(* Logix 5000 project; controller IF2_DEMO Emulate 5570 rev 20.12; software revision 20.04; part 6 of 8 *)
(* tags used below, declared in another part *)
   Alarm_RapidMixStopped : ALARM_DIGITAL;
   CIPSteps : DINT;
   Complete_Manual_Step_AUTO : TIMER;
   Main : MotionVars;
   Mixer_Step_6_AUTORESET : TIMER;
   repeatCIP : BOOL;
   Restart_CIP_Timer_AUTO : TIMER;
   ChangeOver_In_Progress : BOOL;
   Current_Order : STRING;
   DispenserLine : LineData;
   Filler_Stopped : BOOL;
   InitializeDelay : TIMER;
   Labeler_Stopped : BOOL;
   LastOrderCount : DINT;
   LastOrderNumber : STRING;
   ManualCompleted : BOOL;
   MixAgitatorDelayTimer : TIMER;
   MIXCIPStep_DelayTimer : TIMER;
   MixSteps : DINT;   // 1=Initializing 2=Adding Water 3=Wait for manual 4=Agitate 5=xfer 6=cip 7=complete
   MixTransferOutTimer : TIMER;
   MotionSimClr : DINT;
   MotionSimCntr : COUNTER[10];
   MotionSimEn : DINT;
   Next_Product : DINT;
   OEE_Part_Scrap_Old : DINT;
   OEE_Parts_Good_Old : DINT;
   OEE_Parts_Total_Old : DINT;
   OEE_Scrap_Packaging : DINT;
   OrderQty : DINT[4];
   Packaging_Stopped : BOOL;
   PartCountRollOver : DINT;
   Product_Change : DINT;
   Production_Start_Packaging : BOOL;
   ProductionStart : BOOL;
   RapidMixActive : BOOL;
   RapidMixTimer : TIMER;
   RotateTimer : TIMER;
   Starve_Block_Filler_Start_Toggle : BOOL;
   Starve_Block_Labeler_Start_Toggle : BOOL;
   Starve_Block_Packaging_Start_Toggle : BOOL;
   Timer1000ms : TIMER;
   Timer250ms : TIMER;
   WallClock : DINT[7];
   WC : WC[10];
(* Main, continued *)

ROUTINE RapidMix   (* ladder *)
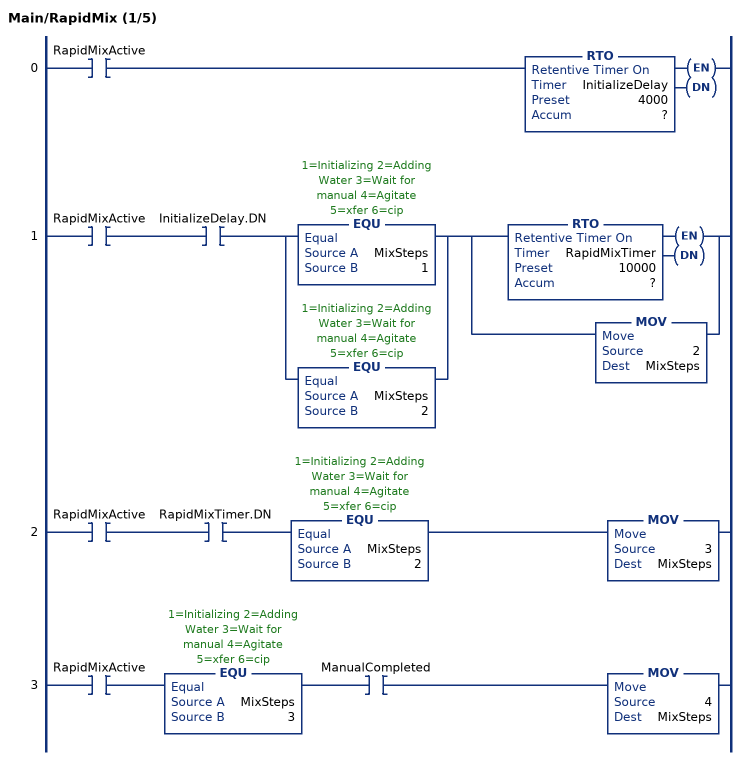
   0: XIC(RapidMixActive)RTO(InitializeDelay,?,?);
   1: XIC(RapidMixActive)XIC(InitializeDelay.DN)[EQU(MixSteps,1) ,EQU(MixSteps,2) ][RTO(RapidMixTimer,?,?) ,MOV(2,MixSteps) ];
   2: XIC(RapidMixActive)XIC(RapidMixTimer.DN)EQU(MixSteps,2)MOV(3,MixSteps);
   3: XIC(RapidMixActive)EQU(MixSteps,3)XIC(ManualCompleted)MOV(4,MixSteps);
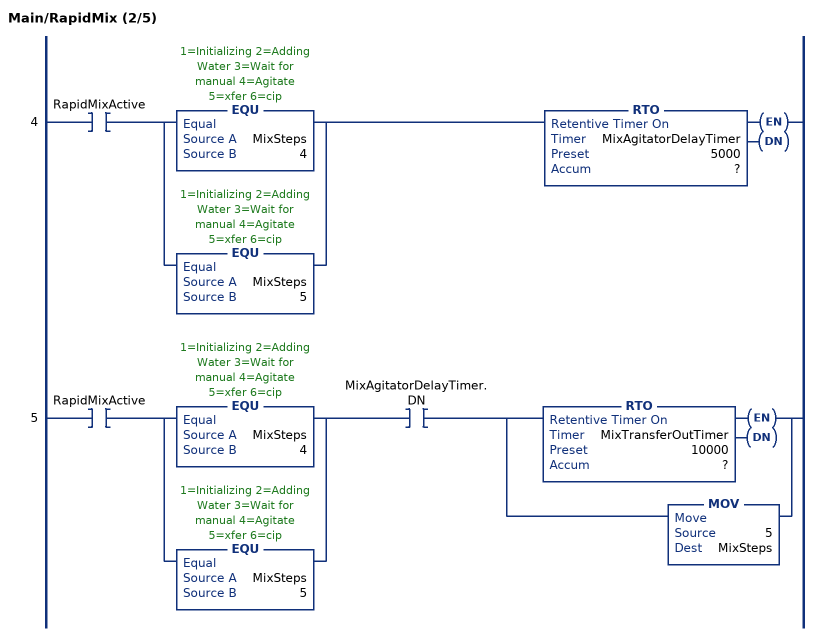
   4: XIC(RapidMixActive)[EQU(MixSteps,4) ,EQU(MixSteps,5) ]RTO(MixAgitatorDelayTimer,?,?);
   5: XIC(RapidMixActive)[EQU(MixSteps,4) ,EQU(MixSteps,5) ]XIC(MixAgitatorDelayTimer.DN)[RTO(MixTransferOutTimer,?,?) ,MOV(5,MixSteps) ];
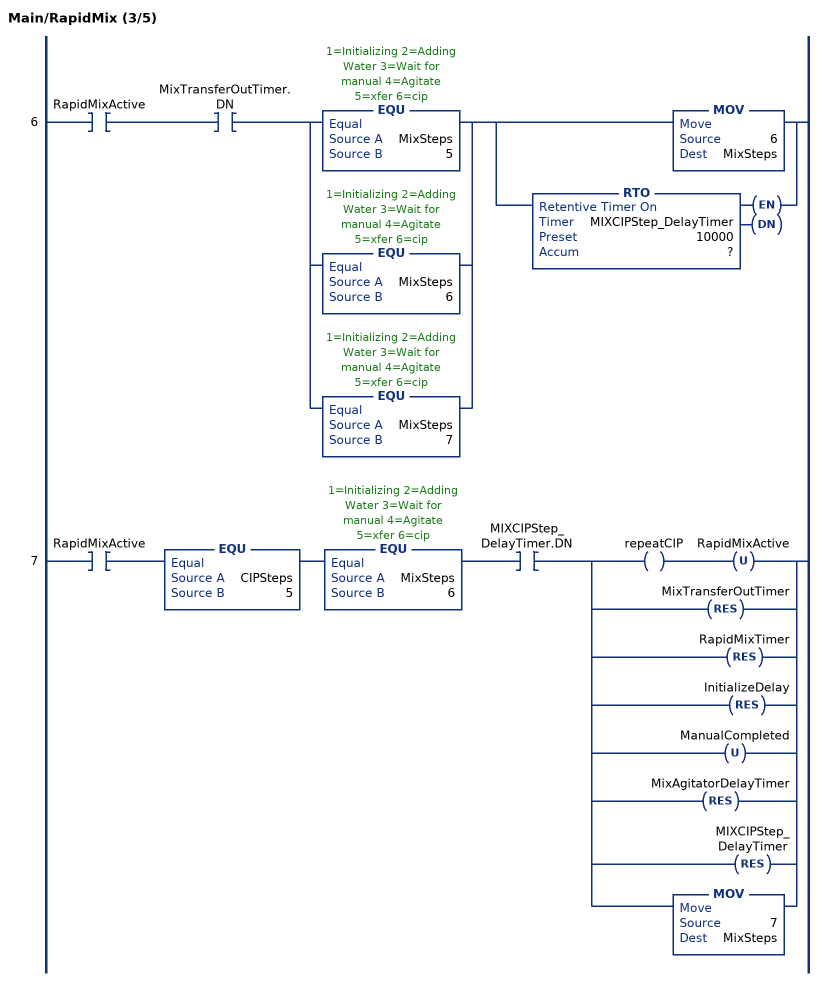
   6: XIC(RapidMixActive)XIC(MixTransferOutTimer.DN)[EQU(MixSteps,5) ,EQU(MixSteps,6) ,EQU(MixSteps,7) ][MOV(6,MixSteps) ,RTO(MIXCIPStep_DelayTimer,?,?) ];
   7: XIC(RapidMixActive)EQU(CIPSteps,5)EQU(MixSteps,6)XIC(MIXCIPStep_DelayTimer.DN)[OTE(repeatCIP) OTU(RapidMixActive) ,[RES(MixTransferOutTimer) ,RES(RapidMixTimer) ,RES(InitializeDelay) ,OTU(ManualCompleted) ,RES(MixAgitatorDelayTimer) ,RES(MIXCIPStep_DelayTimer) ,MOV(7,MixSteps) ] ];
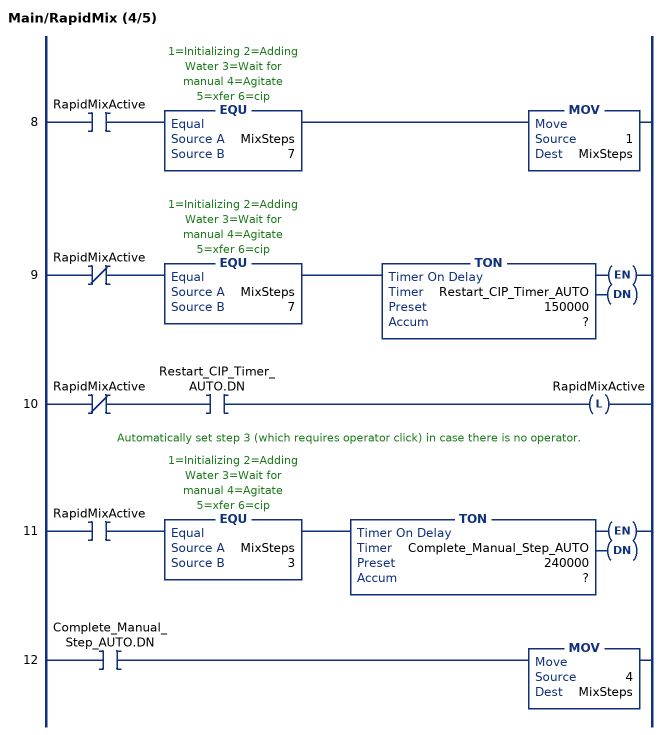
   8: XIC(RapidMixActive)EQU(MixSteps,7)MOV(1,MixSteps);
   9: XIO(RapidMixActive)EQU(MixSteps,7)TON(Restart_CIP_Timer_AUTO,?,?);
   10: XIO(RapidMixActive)XIC(Restart_CIP_Timer_AUTO.DN)OTL(RapidMixActive);
   // Automatically set step 3 (which requires operator click) in case there is no operator.
   11: XIC(RapidMixActive)EQU(MixSteps,3)TON(Complete_Manual_Step_AUTO,?,?);
   12: XIC(Complete_Manual_Step_AUTO.DN)MOV(4,MixSteps);
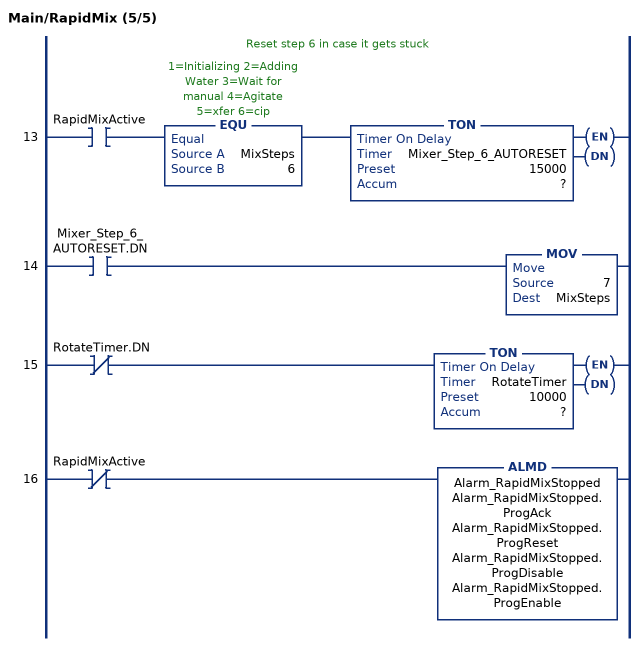
   // Reset step 6 in case it gets stuck
   13: XIC(RapidMixActive)EQU(MixSteps,6)TON(Mixer_Step_6_AUTORESET,?,?);
   14: XIC(Mixer_Step_6_AUTORESET.DN)MOV(7,MixSteps);
   15: XIO(RotateTimer.DN)TON(RotateTimer,?,?);
   16: XIO(RapidMixActive)ALMD(Alarm_RapidMixStopped,Alarm_RapidMixStopped.ProgAck,Alarm_RapidMixStopped.ProgReset,Alarm_RapidMixStopped.ProgDisable,Alarm_RapidMixStopped.ProgEnable);
END_ROUTINE
END_PROGRAM

PROGRAM MotionProg   (* main routine MotionSim *)

ROUTINE MotionSim   (* ladder *)
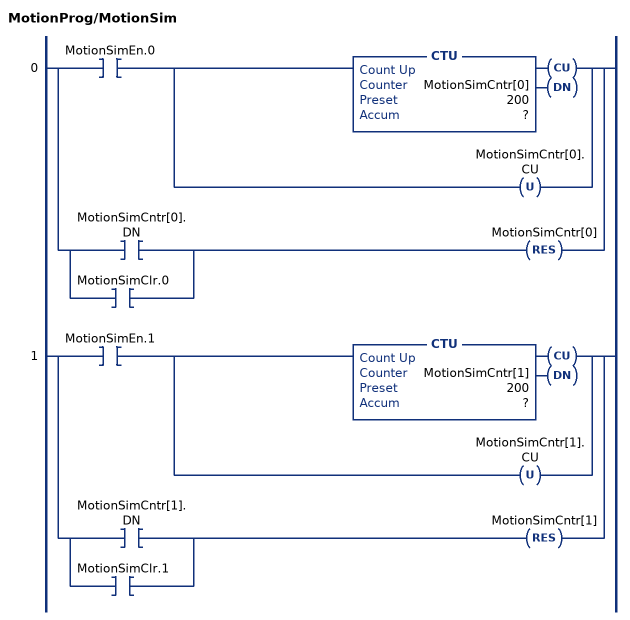
   0: [XIC(MotionSimEn.0) [CTU(MotionSimCntr[0],?,?) ,OTU(MotionSimCntr[0].CU) ] ,[XIC(MotionSimCntr[0].DN) ,XIC(MotionSimClr.0) ] RES(MotionSimCntr[0]) ];
   1: [XIC(MotionSimEn.1) [CTU(MotionSimCntr[1],?,?) ,OTU(MotionSimCntr[1].CU) ] ,[XIC(MotionSimCntr[1].DN) ,XIC(MotionSimClr.1) ] RES(MotionSimCntr[1]) ];
END_ROUTINE
END_PROGRAM

PROGRAM PackD   (* main routine MainRoutine *)
VAR
   Alarm_Packer1_Blocked : ALARM_DIGITAL;
   Alarm_Packer1_Starved : ALARM_DIGITAL;
   Alarm_Packer1_Stopped : ALARM_DIGITAL;
   ATest : BOOL;
   Block_Delay : TIMER := (PRE := 15000);
   Blocked_L : BOOL;
   BottleNum : STRING := '3';
   Ctrl_Bit : BOOL;
   Current_OEE_Availability : REAL := 0.91280067;
   Current_OEE_Availability_MUL100 : DINT := 91;
   Current_OEE_Available : REAL := 58573.0;
   Current_OEE_AvailableTimer : TIMER := (PRE := 3600000, ACC := 58573, EN := 1, TT := 1);
   Current_OEE_Ideal_Cycle : DINT;
   Current_OEE_Overall : REAL := 0.6272021;
   Current_OEE_Performance : REAL := 0.7758806;
   Current_OEE_Performance_MUL100 : DINT := 78;
   Current_OEE_Quality : REAL := 0.8855981;
   Current_OEE_Quality_MUL100 : DINT := 89;
   Current_OEE_Running : REAL := 53545.0;
   Current_OEE_RunningTimer : TIMER := (PRE := 3600000, ACC := 53545, EN := 1, TT := 1);
   DownStream_Run : BOOL := 1;   // Not used - no downstream wc
   DownStream_Running : BOOL := 1;   // Not used - no downstream wc
   Events : Events := (DownTime.Breakdown := 1, DownTime.BreakdownCode := 4, Control.StandbyCode := 1, Control.Auto := 1);
   Events_Control_Auto : ALIAS FOR WC_L.EventTrigger[0].5;
   Events_Control_OpStop : ALIAS FOR WC_L.EventTrigger[0].3;
   Events_Control_Run : ALIAS FOR WC_L.EventTrigger[0].1;
   Events_Control_Running : BOOL := 1;
   Events_Control_Standby : ALIAS FOR WC_L.EventTrigger[0].0;
   Events_Control_StandbyCode : ALIAS FOR WC_L.EventValue_REAL[1];
   Events_DownTime_Breakdown : ALIAS FOR WC_L.EventTrigger[0].2;
   Events_DownTime_BreakdownCode : ALIAS FOR WC_L.EventValue_REAL[2];
   Events_DownTime_Testing : ALIAS FOR WC_L.EventTrigger[0].7;
   Events_DownTime_UnschedMaint : ALIAS FOR WC_L.EventTrigger[0].6;
   Events_Operate_Load : ALIAS FOR WC_L.EventTrigger[0].10;
   Events_Operate_OrderProc : ALIAS FOR WC_L.EventTrigger[0].11;
   Events_Operate_Setup : ALIAS FOR WC_L.EventTrigger[0].9;
   Expected_Full_Production_Rate : REAL := 116.4;
   Expected_Full_Production_Rate_MAX : REAL := 129.4;
   Filler_Starved : ALARM_DIGITAL;
   FillOunces : INT := 32;
   HMI : HMIVars := (ScrapRate := 3.0, SpeedControl := 400.0, PrevSpeed := 100.0, CurrentProductionRate := 120.0, PartCountRollOver := 9999999, MfgTimeBase := 1, MaxEventDur := 21.0, MinEventDur := 9.0, EventsPerHr := 100, EventDur := 17.800318, RunDur := 17.843248, MinRunDur := 5.0);
   Max_Production_Rate_Reached : BOOL := 1;
   MfgOrders : MfgOrders := (CustomerName := 'Big-Mart', OrderName := 'A123', ProdRate := 60.0, PartName := 'Apple-D12', WorkcellName := 'PackD', PartNameSav := 'Apple-D12');
   MfgOrders_CustomerName : ALIAS FOR WC_L.FlexSTRING[4];
   MfgOrders_OrderName : ALIAS FOR WC_L.FlexSTRING[3];
   MfgOrders_PartName : ALIAS FOR WC_L.FlexSTRING[0];
   Motion : DINT := 96;
   Motion1 : DINT := 93;
   Motion_Count : COUNTER := (PRE := 300, ACC := 76);
   Motion_Counter : DINT := 1;
   Motion_Counter1 : DINT := 1;
   Motion_Speed : DINT := 1;
   Motion_Speed_Old : DINT := 25000;
   MotionCount : TIMER := (PRE := 200, ACC := 96, EN := 1, TT := 1);
   MotionCount1 : TIMER := (PRE := 720);
   OEE : OEE := (IdealCycleTime := 5.0, Parts.Total := 1051, Parts.Good := 998, Parts.Scrap := 53);
   OEE_Availability_Previous_1 : REAL := 0.923863;
   OEE_Availability_Previous_2 : REAL := 0.9347185;
   OEE_Availability_Previous_3 : REAL := 0.9347136;
   OEE_IdealCycleTime : ALIAS FOR WC_L.IdealCT;
   OEE_Overall_Previous_1 : REAL := 0.6488823;
   OEE_Overall_Previous_2 : REAL := 0.6521157;
   OEE_Overall_Previous_3 : REAL := 0.65420514;
   OEE_Parts_Good : ALIAS FOR WC_L.GoodParts;
   OEE_Parts_Scrap : ALIAS FOR WC_L.ScrapParts;
   OEE_Parts_Total : ALIAS FOR WC_L.TotalParts;
   OEE_Performance_Previous_1 : REAL := 0.9016351;
   OEE_Performance_Previous_2 : REAL := 0.9124952;
   OEE_Performance_Previous_3 : REAL := 0.91248894;
   OEE_Quality_Previous_1 : REAL := 0.7789823;
   OEE_Quality_Previous_2 : REAL := 0.7645629;
   OEE_Quality_Previous_3 : REAL := 0.76702195;
   onsbits : DINT;
   OperatorID : ALIAS FOR WC_L.FlexREAL[1];
   OutputTargetTimer : TIMER := (PRE := 500000, ACC := 253215, EN := 1, TT := 1);
   Packagin_Bottler_Per_Min : REAL := 112.64006;
   Packaging_Cases_Good : DINT := 34;
   Packaging_Cases_Motion : DINT := 54;
   Packaging_Cases_Per_Minute : REAL := 1.5644453;
   Packaging_Cases_Rejected : DINT := 1;
   Packaging_Cases_Total : DINT := 35;
   Packaging_Start : BOOL := 1;
   Packaging_Status : DINT := 1;
   Packaging_Stop : BOOL;
   Packer : FTVPDemoWorkCell := (RunState := 1, Temperature := 95, GoodParts := 3397, ScrapParts := 105, ScrapRate := 6, ProductionRate := 119, Pressure := 123, OrderName := 'GF-08-CZ-525', CustomerName := 'Soda Inc.', PartName := 'GF-11');
   Packer_State : DINT;
   Pressure1 : ALIAS FOR WC_L.PV[0];   // PSI
   ProductColor : DINT := 1;
   ProductColorCode : INT;
   RecipeFlag : BOOL;
   RecipeName : STRING := 'Super';
   SIM : SimVars := (Run.PRE := 17843, Event.PRE := 9000, Setup.PRE := 9000, Good := 2426.899, Scrap := 75.06019, EventNumber := 11, UtilityBool[1] := 1, UtilityBool[2] := 1);
        .UTILITYBOOL[0]   // Enter Auto Mode ONS
        .UTILITYBOOL[1]   // Work Order Complete ONS
        .UTILITYBOOL[2]   // First Scan Bit
   Starve_Block_Packaging_ONS : BOOL;
   Starve_Delay : TIMER := (PRE := 15000);
   Starved_Condition : BOOL;
   Starved_L : BOOL;
   StateValue : ALIAS FOR WC_L.MonitorValue[0];
   Steady_Production_Rate : TIMER := (PRE := 22000);
   Suppress : Events;
   Temperature1 : ALIAS FOR WC_L.PV[1];   // DEG
   TempReadTrigger : TIMER := (PRE := 5000, ACC := 3794, EN := 1, TT := 1);
   TempTimer : TIMER := (PRE := 10000, ACC := 3900, EN := 1, TT := 1);
   TempTimer2 : TIMER := (PRE := 5000, ACC := 3794, EN := 1, TT := 1);
   Timer_To_Pack_Changeover : TIMER := (PRE := 30000);
   UpStream_Run : ALIAS FOR WC[4].EventTrigger[0].1;
   UpStream_Running : ALIAS FOR WC[4].EventTrigger[0].8;
   WC_L : ALIAS FOR WC[8];
END_VAR

ROUTINE MainRoutine   (* ladder *)
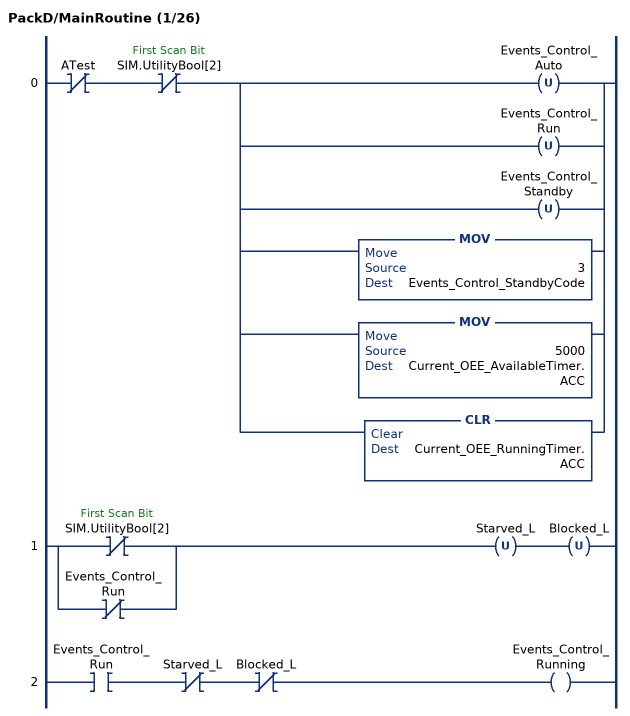
   0: XIO(ATest)XIO(SIM.UtilityBool[2])[OTU(Events_Control_Auto) ,OTU(Events_Control_Run) ,OTU(Events_Control_Standby) ,MOV(3,Events_Control_StandbyCode) ,MOV(5000,Current_OEE_AvailableTimer.ACC) ,CLR(Current_OEE_RunningTimer.ACC) ];
   1: [XIO(SIM.UtilityBool[2]) ,XIO(Events_Control_Run) ]OTU(Starved_L)OTU(Blocked_L);
   2: XIC(Events_Control_Run)XIO(Starved_L)XIO(Blocked_L)OTE(Events_Control_Running);
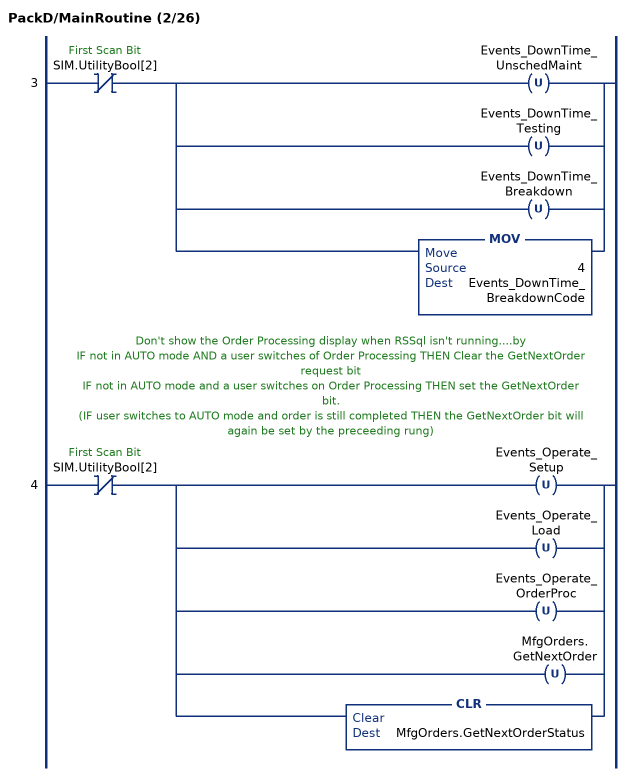
   3: XIO(SIM.UtilityBool[2])[OTU(Events_DownTime_UnschedMaint) ,OTU(Events_DownTime_Testing) ,OTU(Events_DownTime_Breakdown) ,MOV(4,Events_DownTime_BreakdownCode) ];
   // Don't show the Order Processing display when RSSql isn't running....by
   // IF not in AUTO mode AND a user switches of Order Processing THEN Clear the GetNextOrder request bit
   // IF not in AUTO mode and a user switches on Order Processing THEN set the GetNextOrder bit.
   // (IF user switches to AUTO mode and order is still completed THEN the GetNextOrder bit will again be set by the preceeding rung)
   4: XIO(SIM.UtilityBool[2])[OTU(Events_Operate_Setup) ,OTU(Events_Operate_Load) ,OTU(Events_Operate_OrderProc) ,OTU(MfgOrders.GetNextOrder) ,CLR(MfgOrders.GetNextOrderStatus) ];
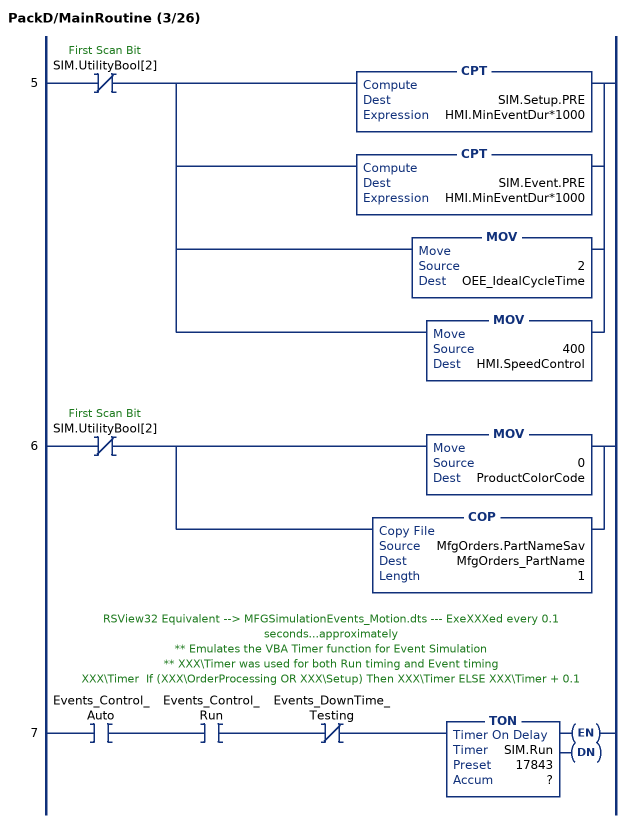
   5: XIO(SIM.UtilityBool[2])[CPT(SIM.Setup.PRE,HMI.MinEventDur*1000) ,CPT(SIM.Event.PRE,HMI.MinEventDur*1000) ,MOV(2,OEE_IdealCycleTime) ,MOV(400,HMI.SpeedControl) ];
   6: XIO(SIM.UtilityBool[2])[MOV(0,ProductColorCode) ,COP(MfgOrders.PartNameSav,MfgOrders_PartName,1) ];
   // RSView32 Equivalent --> MFGSimulationEvents_Motion.dts --- ExeXXXed every 0.1 seconds...approximately
   // ** Emulates the VBA Timer function for Event Simulation
   // ** XXX\Timer was used for both Run timing and Event timing
   // XXX\Timer	If (XXX\OrderProcessing OR XXX\Setup) Then XXX\Timer ELSE XXX\Timer + 0.1
   7: XIC(Events_Control_Auto)XIC(Events_Control_Run)XIO(Events_DownTime_Testing)TON(SIM.Run,?,?);
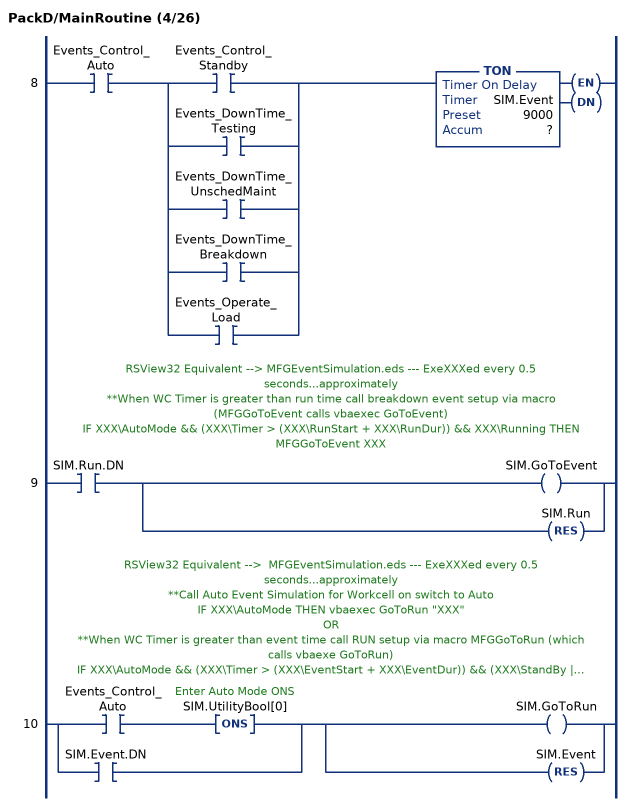
   8: XIC(Events_Control_Auto)[XIC(Events_Control_Standby) ,XIC(Events_DownTime_Testing) ,XIC(Events_DownTime_UnschedMaint) ,XIC(Events_DownTime_Breakdown) ,XIC(Events_Operate_Load) ]TON(SIM.Event,?,?);
   // RSView32 Equivalent --> MFGEventSimulation.eds --- ExeXXXed every 0.5 seconds...approximately
   // **When WC Timer is greater than run time call breakdown event setup via macro (MFGGoToEvent calls vbaexec GoToEvent)
   // IF XXX\AutoMode && (XXX\Timer > (XXX\RunStart + XXX\RunDur)) && XXX\Running THEN MFGGoToEvent XXX
   9: XIC(SIM.Run.DN)[OTE(SIM.GoToEvent) ,RES(SIM.Run) ];
   // RSView32 Equivalent -->  MFGEventSimulation.eds --- ExeXXXed every 0.5 seconds...approximately
   // **Call Auto Event Simulation for Workcell on switch to Auto
   // IF XXX\AutoMode THEN vbaexec GoToRun "XXX"
   // OR
   // **When WC Timer is greater than event time call RUN setup via macro MFGGoToRun (which calls vbaexe GoToRun)
   // IF XXX\AutoMode && (XXX\Timer > (XXX\EventStart + XXX\EventDur)) && (XXX\StandBy || XXX\Test || XXX\UnSchedMaint || XXX\Breakdown ||XXX\Load) THEN MFGGoToRun XXX
   10: [XIC(Events_Control_Auto) ONS(SIM.UtilityBool[0]) ,XIC(SIM.Event.DN) ][OTE(SIM.GoToRun) ,RES(SIM.Event) ];
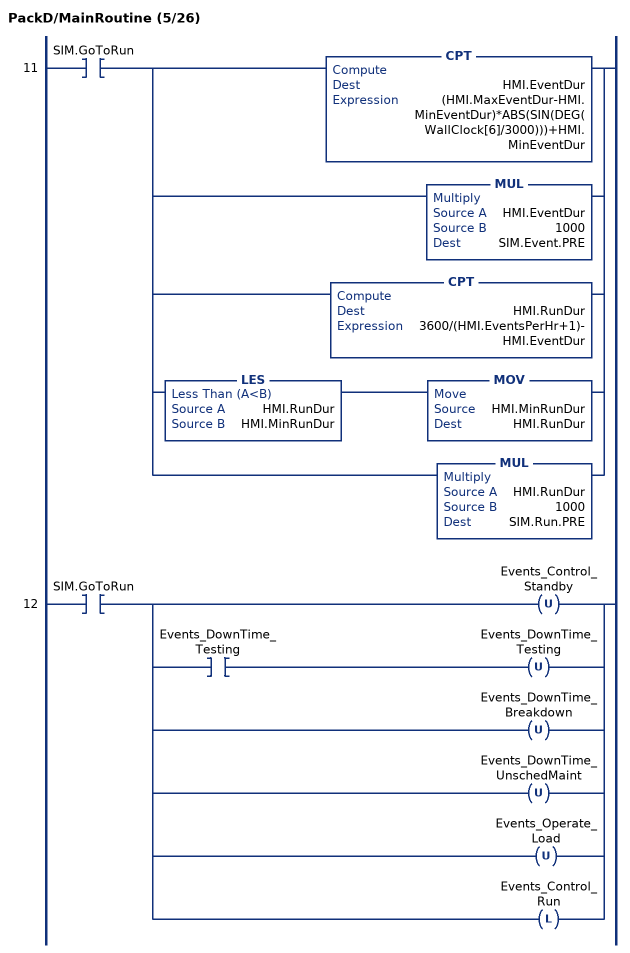
   11: XIC(SIM.GoToRun)[CPT(HMI.EventDur,(HMI.MaxEventDur-HMI.MinEventDur)*ABS(SIN(DEG(WallClock[6]/3000)))+HMI.MinEventDur) ,MUL(HMI.EventDur,1000,SIM.Event.PRE) ,CPT(HMI.RunDur,3600/(HMI.EventsPerHr+1)-HMI.EventDur) ,LES(HMI.RunDur,HMI.MinRunDur) MOV(HMI.MinRunDur,HMI.RunDur) ,MUL(HMI.RunDur,1000,SIM.Run.PRE) ];
   12: XIC(SIM.GoToRun)[OTU(Events_Control_Standby) ,XIC(Events_DownTime_Testing) OTU(Events_DownTime_Testing) ,OTU(Events_DownTime_Breakdown) ,OTU(Events_DownTime_UnschedMaint) ,OTU(Events_Operate_Load) ,OTL(Events_Control_Run) ];
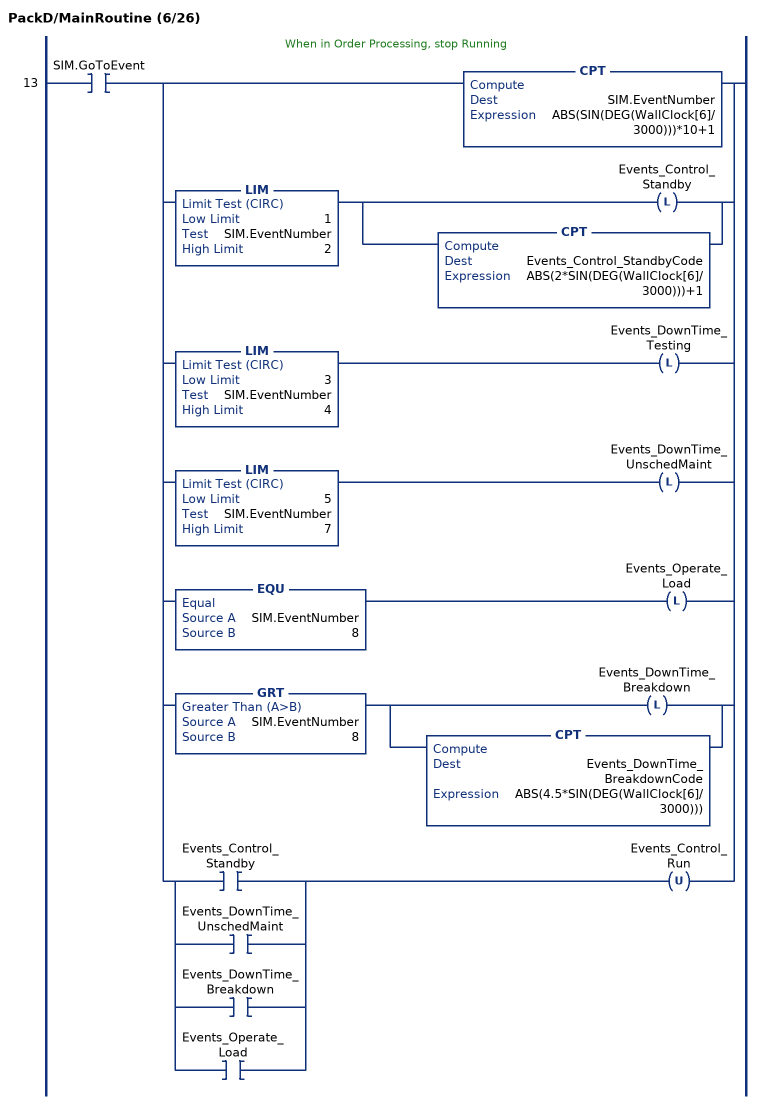
   // When in Order Processing, stop Running
   13: XIC(SIM.GoToEvent)[CPT(SIM.EventNumber,ABS(SIN(DEG(WallClock[6]/3000)))*10+1) ,LIM(1,SIM.EventNumber,2) [OTL(Events_Control_Standby) ,CPT(Events_Control_StandbyCode,ABS(2*SIN(DEG(WallClock[6]/3000)))+1) ] ,LIM(3,SIM.EventNumber,4) OTL(Events_DownTime_Testing) ,LIM(5,SIM.EventNumber,7) OTL(Events_DownTime_UnschedMaint) ,EQU(SIM.EventNumber,8) OTL(Events_Operate_Load) ,GRT(SIM.EventNumber,8) [OTL(Events_DownTime_Breakdown) ,CPT(Events_DownTime_BreakdownCode,ABS(4.5*SIN(DEG(WallClock[6]/3000)))) ] ,[XIC(Events_Control_Standby) ,XIC(Events_DownTime_UnschedMaint) ,XIC(Events_DownTime_Breakdown) ,XIC(Events_Operate_Load) ] OTU(Events_Control_Run) ];
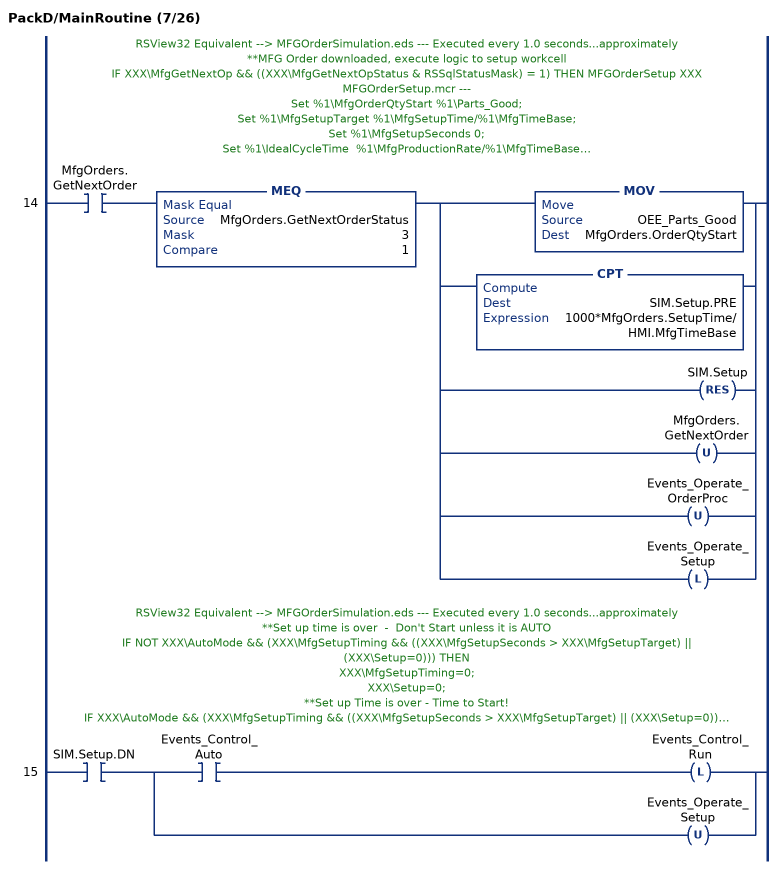
   // RSView32 Equivalent --> MFGOrderSimulation.eds --- Executed every 1.0 seconds...approximately
   // **MFG Order downloaded, execute logic to setup workcell
   // IF XXX\MfgGetNextOp && ((XXX\MfgGetNextOpStatus & RSSqlStatusMask) = 1) THEN MFGOrderSetup XXX
   // MFGOrderSetup.mcr ---
   // 	Set %1\MfgOrderQtyStart %1\Parts_Good;
   // 	Set %1\MfgSetupTarget %1\MfgSetupTime/%1\MfgTimeBase;
   // 	Set %1\MfgSetupSeconds 0;
   // 	Set %1\IdealCycleTime  %1\MfgProductionRate/%1\MfgTimeBase;
   // 	Set %1\MfgGetNextOp 0;
   // 	Set %1\Setup 1;
   // 	Set %1\OrderProcessing 0;
   // 	Set %1\MfgSetupTiming 1;
   14: XIC(MfgOrders.GetNextOrder)MEQ(MfgOrders.GetNextOrderStatus,3,1)[MOV(OEE_Parts_Good,MfgOrders.OrderQtyStart) ,CPT(SIM.Setup.PRE,1000*MfgOrders.SetupTime/HMI.MfgTimeBase) ,RES(SIM.Setup) ,OTU(MfgOrders.GetNextOrder) ,OTU(Events_Operate_OrderProc) ,OTL(Events_Operate_Setup) ];
   // RSView32 Equivalent --> MFGOrderSimulation.eds --- Executed every 1.0 seconds...approximately
   // **Set up time is over  -  Don't Start unless it is AUTO
   // IF NOT XXX\AutoMode && (XXX\MfgSetupTiming && ((XXX\MfgSetupSeconds > XXX\MfgSetupTarget) || (XXX\Setup=0))) THEN
   // 	XXX\MfgSetupTiming=0;
   // 	XXX\Setup=0;
   // **Set up Time is over - Time to Start!
   // IF XXX\AutoMode && (XXX\MfgSetupTiming && ((XXX\MfgSetupSeconds > XXX\MfgSetupTarget) || (XXX\Setup=0))) THEN
   // 	XXX\MfgSetupTiming=0;
   // 	XXX\Setup=0;
   // 	XXX\RUNNING=1
   15: XIC(SIM.Setup.DN)[XIC(Events_Control_Auto) OTL(Events_Control_Run) ,OTU(Events_Operate_Setup) ];
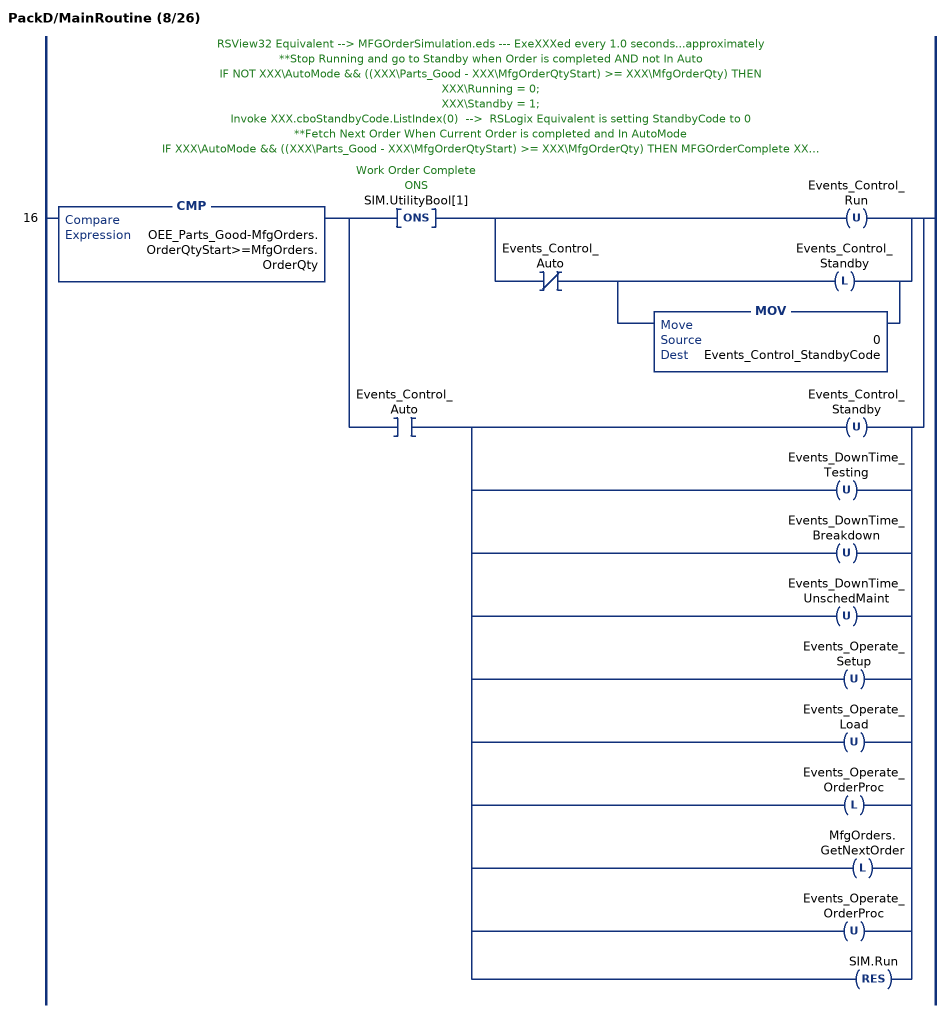
   // RSView32 Equivalent --> MFGOrderSimulation.eds --- ExeXXXed every 1.0 seconds...approximately
   // **Stop Running and go to Standby when Order is completed AND not In Auto
   // IF NOT XXX\AutoMode && ((XXX\Parts_Good - XXX\MfgOrderQtyStart) >= XXX\MfgOrderQty) THEN
   // 	XXX\Running = 0;
   // 	XXX\Standby = 1;
   // 	Invoke XXX.cboStandbyCode.ListIndex(0)  -->  RSLogix Equivalent is setting StandbyCode to 0
   // **Fetch Next Order When Current Order is completed and In AutoMode
   // IF XXX\AutoMode && ((XXX\Parts_Good - XXX\MfgOrderQtyStart) >= XXX\MfgOrderQty) THEN MFGOrderComplete XXX
   // MFGOrderComplete.mcr --- (Macros exeXXXed when called. %1 is the Workcell name -- typical all mcrs)
   // 	Set %1\RunStart %1\Timer;
   // 	Set %1\StandBy 0;
   // 	Set %1\Test 0;
   // 	Set %1\UnSchedMaint 0;
   // 	Set %1\Breakdown 0;
   // 	Set %1\Load 0;
   // 	Set %1\OrderProcessing 1;
   // 	Set %1\Running 0;
   // 	Set %1\MFGGetNextOpStatus 0;
   // 	Set %1\MFGGetNextOp 1
   16: CMP(OEE_Parts_Good-MfgOrders.OrderQtyStart>=MfgOrders.OrderQty)[ONS(SIM.UtilityBool[1]) [OTU(Events_Control_Run) ,XIO(Events_Control_Auto) [OTL(Events_Control_Standby) ,MOV(0,Events_Control_StandbyCode) ] ] ,XIC(Events_Control_Auto) [OTU(Events_Control_Standby) ,OTU(Events_DownTime_Testing) ,OTU(Events_DownTime_Breakdown) ,OTU(Events_DownTime_UnschedMaint) ,OTU(Events_Operate_Setup) ,OTU(Events_Operate_Load) ,OTL(Events_Operate_OrderProc) ,OTL(MfgOrders.GetNextOrder) ,OTU(Events_Operate_OrderProc) ,RES(SIM.Run) ] ];
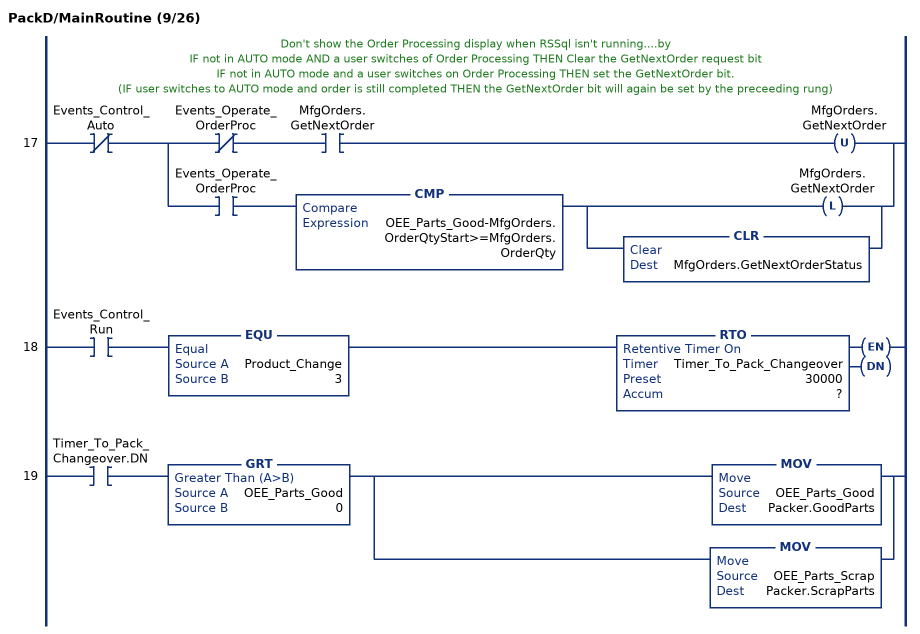
   // Don't show the Order Processing display when RSSql isn't running....by
   // IF not in AUTO mode AND a user switches of Order Processing THEN Clear the GetNextOrder request bit
   // IF not in AUTO mode and a user switches on Order Processing THEN set the GetNextOrder bit.
   // (IF user switches to AUTO mode and order is still completed THEN the GetNextOrder bit will again be set by the preceeding rung)
   17: XIO(Events_Control_Auto)[XIO(Events_Operate_OrderProc) XIC(MfgOrders.GetNextOrder) OTU(MfgOrders.GetNextOrder) ,XIC(Events_Operate_OrderProc) CMP(OEE_Parts_Good-MfgOrders.OrderQtyStart>=MfgOrders.OrderQty) [OTL(MfgOrders.GetNextOrder) ,CLR(MfgOrders.GetNextOrderStatus) ] ];
   18: XIC(Events_Control_Run)EQU(Product_Change,3)RTO(Timer_To_Pack_Changeover,?,?);
   19: XIC(Timer_To_Pack_Changeover.DN)GRT(OEE_Parts_Good,0)[MOV(OEE_Parts_Good,Packer.GoodParts) ,MOV(OEE_Parts_Scrap,Packer.ScrapParts) ];
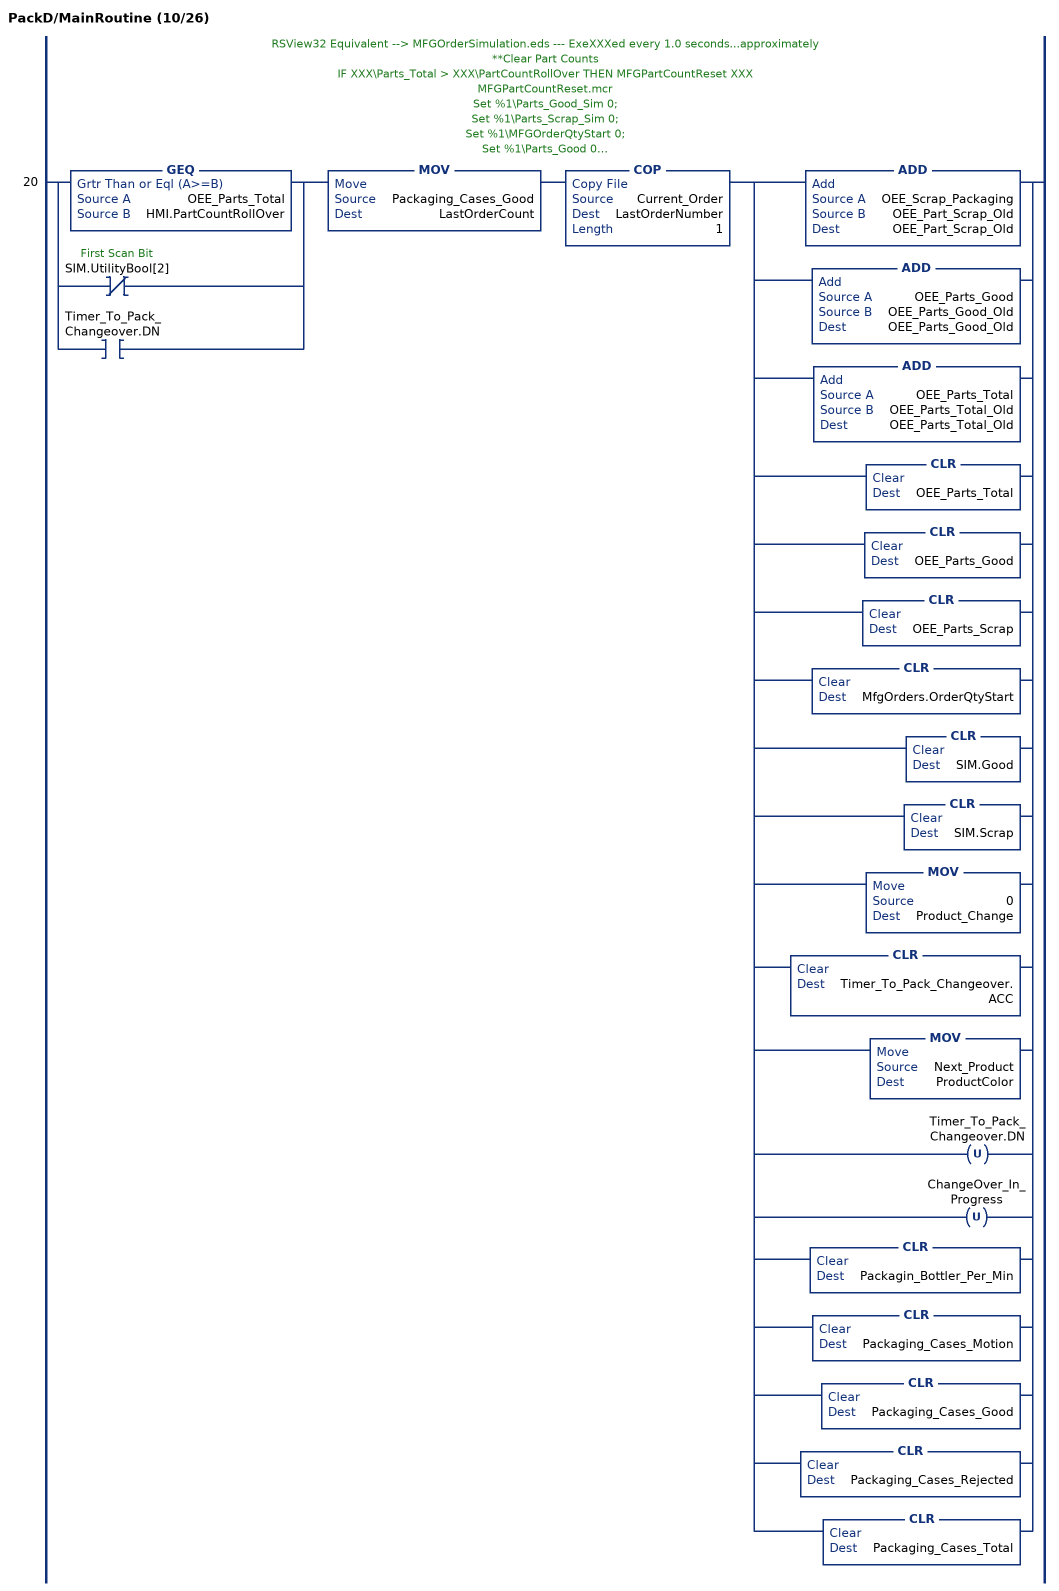
   // RSView32 Equivalent --> MFGOrderSimulation.eds --- ExeXXXed every 1.0 seconds...approximately
   // **Clear Part Counts
   // IF XXX\Parts_Total > XXX\PartCountRollOver THEN MFGPartCountReset XXX
   // MFGPartCountReset.mcr
   // 	Set %1\Parts_Good_Sim 0;
   // 	Set %1\Parts_Scrap_Sim 0;
   // 	Set %1\MFGOrderQtyStart 0;
   // 	Set %1\Parts_Good 0;
   // 	Set %1\Parts_Scrap 0;
   // 	Set %1\Parts_Total 0
   20: [GEQ(OEE_Parts_Total,HMI.PartCountRollOver) ,XIO(SIM.UtilityBool[2]) ,XIC(Timer_To_Pack_Changeover.DN) ]MOV(Packaging_Cases_Good,LastOrderCount)COP(Current_Order,LastOrderNumber,1)[ADD(OEE_Scrap_Packaging,OEE_Part_Scrap_Old,OEE_Part_Scrap_Old) ,ADD(OEE_Parts_Good,OEE_Parts_Good_Old,OEE_Parts_Good_Old) ,ADD(OEE_Parts_Total,OEE_Parts_Total_Old,OEE_Parts_Total_Old) ,CLR(OEE_Parts_Total) ,CLR(OEE_Parts_Good) ,CLR(OEE_Parts_Scrap) ,CLR(MfgOrders.OrderQtyStart) ,CLR(SIM.Good) ,CLR(SIM.Scrap) ,MOV(0,Product_Change) ,CLR(Timer_To_Pack_Changeover.ACC) ,MOV(Next_Product,ProductColor) ,OTU(Timer_To_Pack_Changeover.DN) ,OTU(ChangeOver_In_Progress) ,CLR(Packagin_Bottler_Per_Min) ,CLR(Packaging_Cases_Motion) ,CLR(Packaging_Cases_Good) ,CLR(Packaging_Cases_Rejected) ,CLR(Packaging_Cases_Total) ];
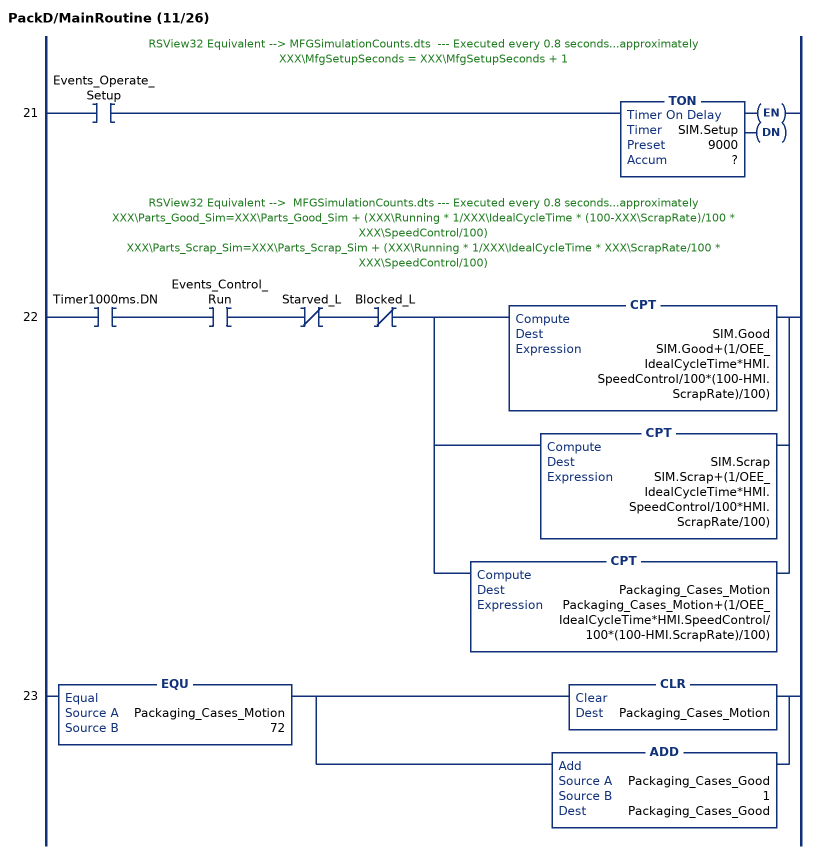
   // RSView32 Equivalent --> MFGSimulationCounts.dts	--- Executed every 0.8 seconds...approximately
   // XXX\MfgSetupSeconds = XXX\MfgSetupSeconds + 1
   21: XIC(Events_Operate_Setup)TON(SIM.Setup,?,?);
   // RSView32 Equivalent -->  MFGSimulationCounts.dts --- Executed every 0.8 seconds...approximately
   // XXX\Parts_Good_Sim=XXX\Parts_Good_Sim + (XXX\Running * 1/XXX\IdealCycleTime * (100-XXX\ScrapRate)/100 * XXX\SpeedControl/100)
   // XXX\Parts_Scrap_Sim=XXX\Parts_Scrap_Sim + (XXX\Running * 1/XXX\IdealCycleTime * XXX\ScrapRate/100 * XXX\SpeedControl/100)
   22: XIC(Timer1000ms.DN)XIC(Events_Control_Run)XIO(Starved_L)XIO(Blocked_L)[CPT(SIM.Good,SIM.Good+(1/OEE_IdealCycleTime*HMI.SpeedControl/100*(100-HMI.ScrapRate)/100)) ,CPT(SIM.Scrap,SIM.Scrap+(1/OEE_IdealCycleTime*HMI.SpeedControl/100*HMI.ScrapRate/100)) ,CPT(Packaging_Cases_Motion,Packaging_Cases_Motion+(1/OEE_IdealCycleTime*HMI.SpeedControl/100*(100-HMI.ScrapRate)/100)) ];
   23: EQU(Packaging_Cases_Motion,72)[CLR(Packaging_Cases_Motion) ,ADD(Packaging_Cases_Good,1,Packaging_Cases_Good) ];
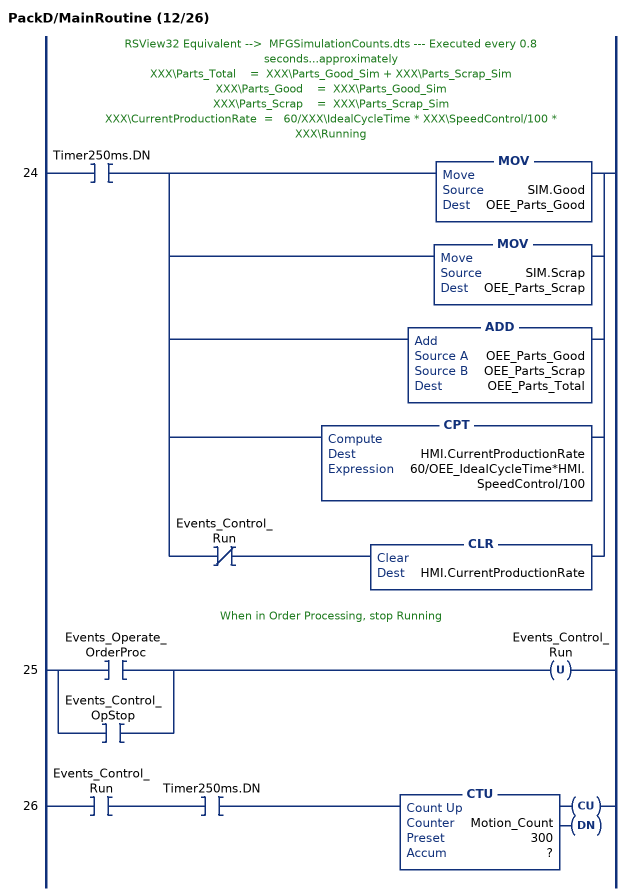
   // RSView32 Equivalent -->  MFGSimulationCounts.dts --- Executed every 0.8 seconds...approximately
   // XXX\Parts_Total		=	XXX\Parts_Good_Sim + XXX\Parts_Scrap_Sim
   // XXX\Parts_Good		=	XXX\Parts_Good_Sim
   // XXX\Parts_Scrap		=	XXX\Parts_Scrap_Sim
   // XXX\CurrentProductionRate  = 	60/XXX\IdealCycleTime * XXX\SpeedControl/100 * XXX\Running
   24: XIC(Timer250ms.DN)[[MOV(SIM.Good,OEE_Parts_Good) ,MOV(SIM.Scrap,OEE_Parts_Scrap) ,ADD(OEE_Parts_Good,OEE_Parts_Scrap,OEE_Parts_Total) ] ,CPT(HMI.CurrentProductionRate,60/OEE_IdealCycleTime*HMI.SpeedControl/100) ,XIO(Events_Control_Run) CLR(HMI.CurrentProductionRate) ];
   // When in Order Processing, stop Running
   25: [XIC(Events_Operate_OrderProc) ,XIC(Events_Control_OpStop) ]OTU(Events_Control_Run);
   26: XIC(Events_Control_Run)XIC(Timer250ms.DN)CTU(Motion_Count,?,?);
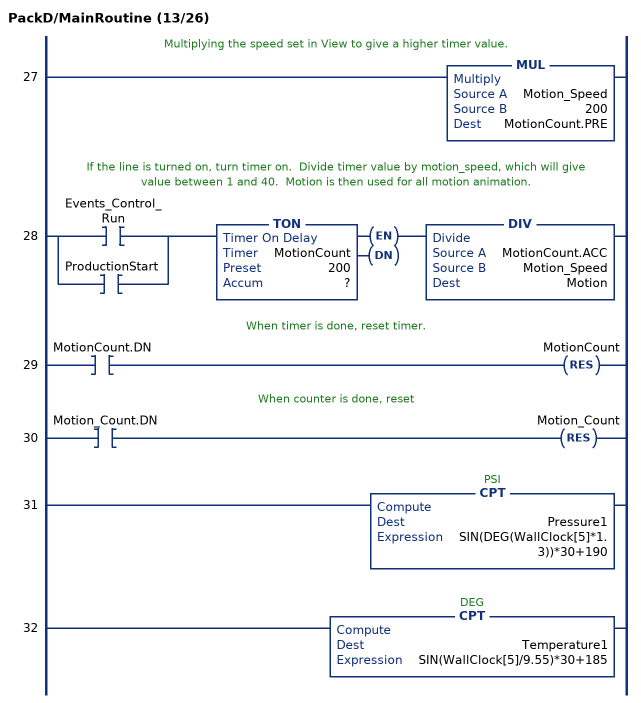
   // Multiplying the speed set in View to give a higher timer value.
   27: MUL(Motion_Speed,200,MotionCount.PRE);
   // If the line is turned on, turn timer on.  Divide timer value by motion_speed, which will give value between 1 and 40.  Motion is then used for all motion animation.
   28: [XIC(Events_Control_Run) ,XIC(ProductionStart) ]TON(MotionCount,?,?)DIV(MotionCount.ACC,Motion_Speed,Motion);
   // When timer is done, reset timer.
   29: XIC(MotionCount.DN)RES(MotionCount);
   // When counter is done, reset
   30: XIC(Motion_Count.DN)RES(Motion_Count);
   31: CPT(Pressure1,SIN(DEG(WallClock[5]*1.3))*30+190);
   32: CPT(Temperature1,SIN(WallClock[5]/9.55)*30+185);
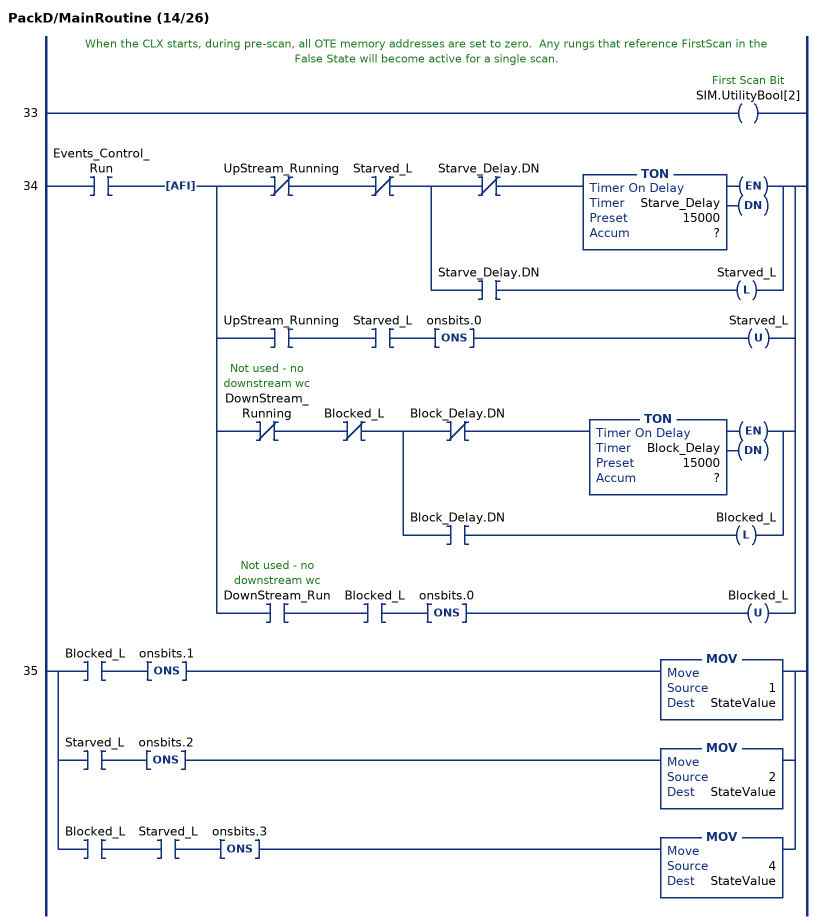
   // When the CLX starts, during pre-scan, all OTE memory addresses are set to zero.  Any rungs that reference FirstScan in the False State will become active for a single scan.
   33: OTE(SIM.UtilityBool[2]);
   34: XIC(Events_Control_Run)AFI()[[XIO(UpStream_Running) XIO(Starved_L) [XIO(Starve_Delay.DN) TON(Starve_Delay,?,?) ,XIC(Starve_Delay.DN) OTL(Starved_L) ] ,XIC(UpStream_Running) XIC(Starved_L) ONS(onsbits.0) OTU(Starved_L) ] ,[XIO(DownStream_Running) XIO(Blocked_L) [XIO(Block_Delay.DN) TON(Block_Delay,?,?) ,XIC(Block_Delay.DN) OTL(Blocked_L) ] ,XIC(DownStream_Run) XIC(Blocked_L) ONS(onsbits.0) OTU(Blocked_L) ] ];
   35: [XIC(Blocked_L) ONS(onsbits.1) MOV(1,StateValue) ,XIC(Starved_L) ONS(onsbits.2) MOV(2,StateValue) ,XIC(Blocked_L) XIC(Starved_L) ONS(onsbits.3) MOV(4,StateValue) ];
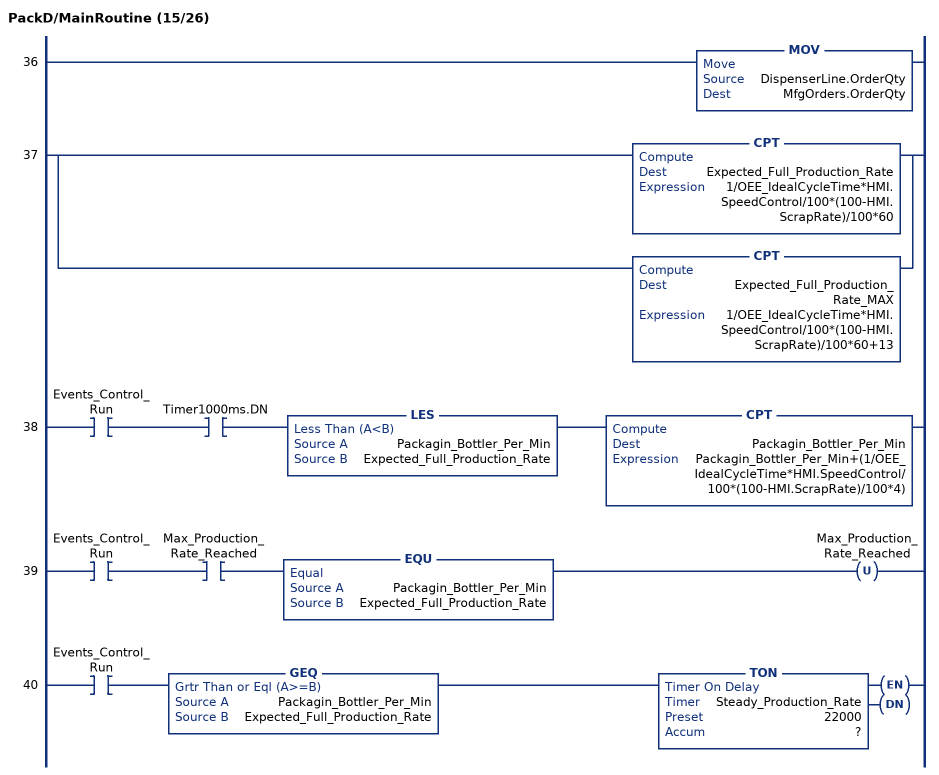
   36: MOV(DispenserLine.OrderQty,MfgOrders.OrderQty);
   37: [CPT(Expected_Full_Production_Rate,1/OEE_IdealCycleTime*HMI.SpeedControl/100*(100-HMI.ScrapRate)/100*60) ,CPT(Expected_Full_Production_Rate_MAX,1/OEE_IdealCycleTime*HMI.SpeedControl/100*(100-HMI.ScrapRate)/100*60+13) ];
   38: XIC(Events_Control_Run)XIC(Timer1000ms.DN)LES(Packagin_Bottler_Per_Min,Expected_Full_Production_Rate)CPT(Packagin_Bottler_Per_Min,Packagin_Bottler_Per_Min+(1/OEE_IdealCycleTime*HMI.SpeedControl/100*(100-HMI.ScrapRate)/100*4));
   39: XIC(Events_Control_Run)XIC(Max_Production_Rate_Reached)EQU(Packagin_Bottler_Per_Min,Expected_Full_Production_Rate)OTU(Max_Production_Rate_Reached);
   40: XIC(Events_Control_Run)GEQ(Packagin_Bottler_Per_Min,Expected_Full_Production_Rate)TON(Steady_Production_Rate,?,?);
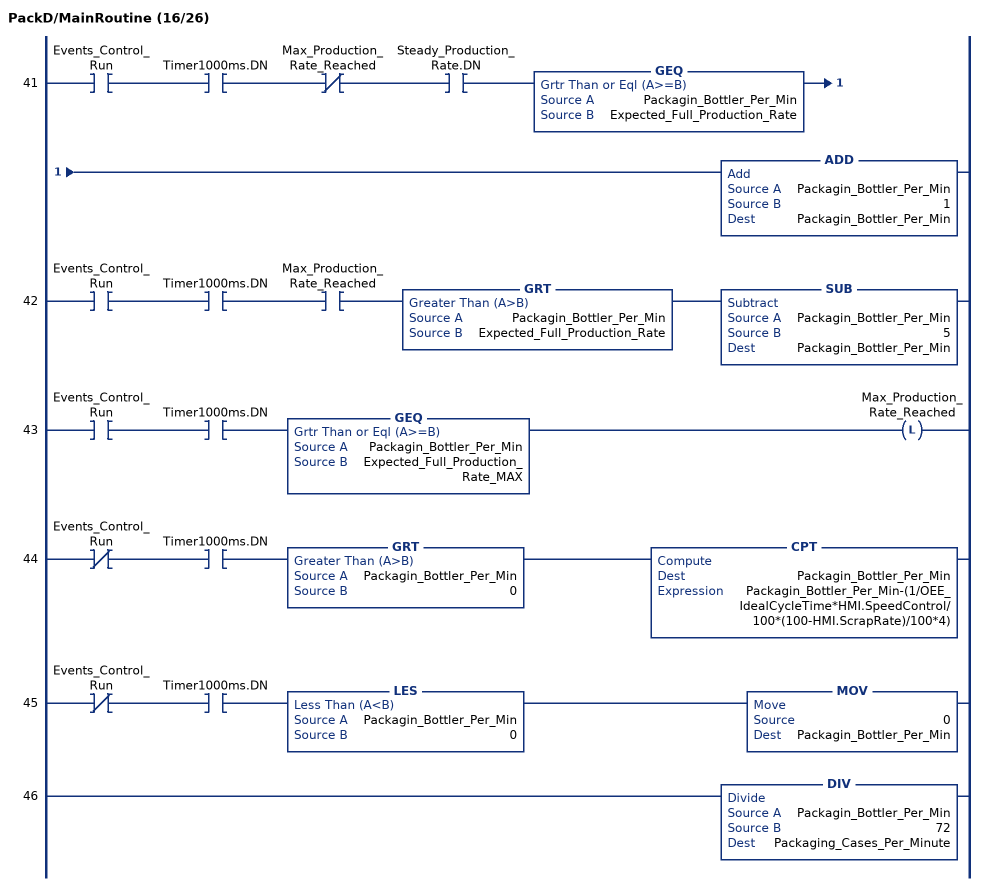
   41: XIC(Events_Control_Run)XIC(Timer1000ms.DN)XIO(Max_Production_Rate_Reached)XIC(Steady_Production_Rate.DN)GEQ(Packagin_Bottler_Per_Min,Expected_Full_Production_Rate)ADD(Packagin_Bottler_Per_Min,1,Packagin_Bottler_Per_Min);
   42: XIC(Events_Control_Run)XIC(Timer1000ms.DN)XIC(Max_Production_Rate_Reached)GRT(Packagin_Bottler_Per_Min,Expected_Full_Production_Rate)SUB(Packagin_Bottler_Per_Min,5,Packagin_Bottler_Per_Min);
   43: XIC(Events_Control_Run)XIC(Timer1000ms.DN)GEQ(Packagin_Bottler_Per_Min,Expected_Full_Production_Rate_MAX)OTL(Max_Production_Rate_Reached);
   44: XIO(Events_Control_Run)XIC(Timer1000ms.DN)GRT(Packagin_Bottler_Per_Min,0)CPT(Packagin_Bottler_Per_Min,Packagin_Bottler_Per_Min-(1/OEE_IdealCycleTime*HMI.SpeedControl/100*(100-HMI.ScrapRate)/100*4));
   45: XIO(Events_Control_Run)XIC(Timer1000ms.DN)LES(Packagin_Bottler_Per_Min,0)MOV(0,Packagin_Bottler_Per_Min);
   46: DIV(Packagin_Bottler_Per_Min,72,Packaging_Cases_Per_Minute);
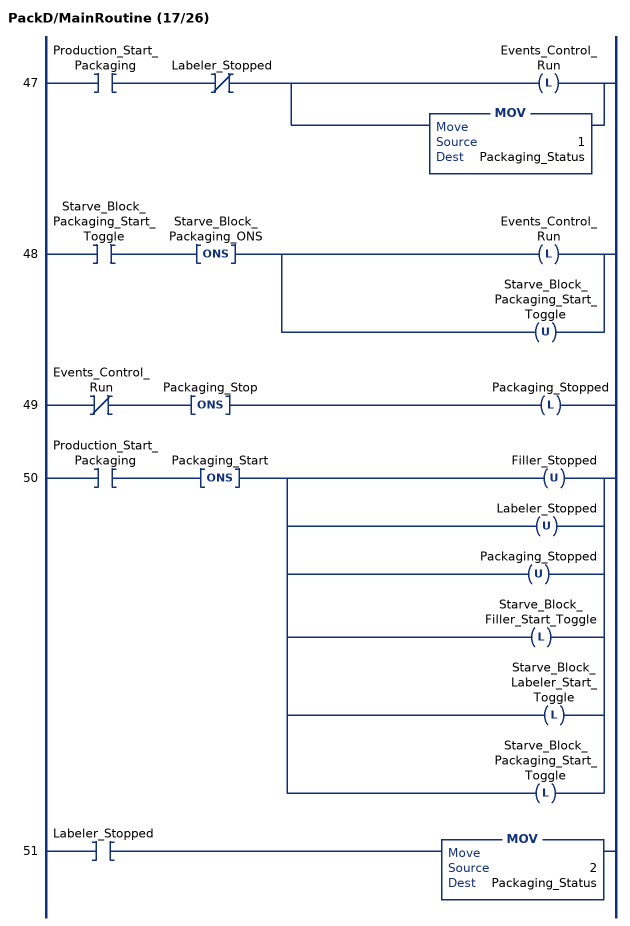
   47: XIC(Production_Start_Packaging)XIO(Labeler_Stopped)[OTL(Events_Control_Run) ,MOV(1,Packaging_Status) ];
   48: XIC(Starve_Block_Packaging_Start_Toggle)ONS(Starve_Block_Packaging_ONS)[OTL(Events_Control_Run) ,OTU(Starve_Block_Packaging_Start_Toggle) ];
   49: XIO(Events_Control_Run)ONS(Packaging_Stop)OTL(Packaging_Stopped);
   50: XIC(Production_Start_Packaging)ONS(Packaging_Start)[OTU(Filler_Stopped) ,OTU(Labeler_Stopped) ,OTU(Packaging_Stopped) ,OTL(Starve_Block_Filler_Start_Toggle) ,OTL(Starve_Block_Labeler_Start_Toggle) ,OTL(Starve_Block_Packaging_Start_Toggle) ];
   51: XIC(Labeler_Stopped)MOV(2,Packaging_Status);
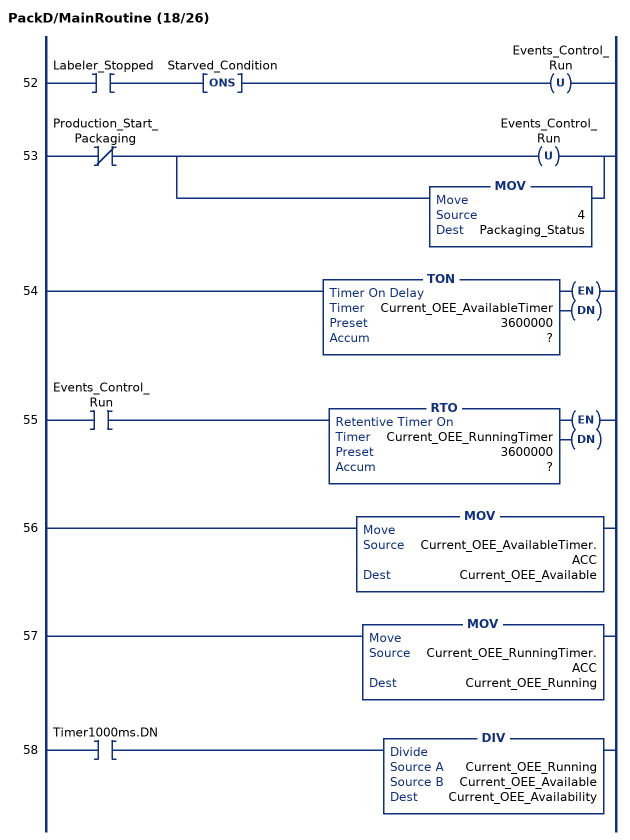
   52: XIC(Labeler_Stopped)ONS(Starved_Condition)OTU(Events_Control_Run);
   53: XIO(Production_Start_Packaging)[OTU(Events_Control_Run) ,MOV(4,Packaging_Status) ];
   54: TON(Current_OEE_AvailableTimer,?,?);
   55: XIC(Events_Control_Run)RTO(Current_OEE_RunningTimer,?,?);
   56: MOV(Current_OEE_AvailableTimer.ACC,Current_OEE_Available);
   57: MOV(Current_OEE_RunningTimer.ACC,Current_OEE_Running);
   58: XIC(Timer1000ms.DN)DIV(Current_OEE_Running,Current_OEE_Available,Current_OEE_Availability);
